FUNCTION_BLOCK FB_DriveInverter EXTENDS FB_DriveReverse IMPLEMENTS I_DriveInverter;
VAR
	_stInverter : ST_Inverter;
			
END_VAR

VAR_STAT
	_nInstances		: INT;		// Counter of created Instances
END_VAR

PROPERTY DeviceData : ST_Inverter
GET
// Dane pobierane i ustawiane podczas obsługi Invertera przez ModbusRtu
DeviceData := _stInverter;
END_GET
END_PROPERTY

METHOD FB_init : BOOL
VAR_INPUT
	bInitRetains : BOOL; // if TRUE, the retain variables are initialized (warm start / cold start)
	bInCopyCode : BOOL;  // if TRUE, the instance afterwards gets moved into the copy code (online change)
	bDeviceId		 : BYTE;	
END_VAR
THIS^._stInverter.bDeviceID := bDeviceID;

//count of FB Instances and setting int Array of Interface variables. Assign an object to an interface variable
// The array of interface variable must be global
_nInstances := _nInstances + 1;
Itf.aItfDriveInverter[_nInstances] := THIS^;
END_METHOD

PROPERTY InstanceCounter : INT
GET
InstanceCounter := _nInstances;
END_GET
END_PROPERTY

METHOD Reset : BOOL
VAR_INPUT
END_VAR


// Set reset Command
THIS^._stInverter.eControl := eReset;
END_METHOD

METHOD SetSpeed : BOOL
VAR_INPUT
	_speed	: REAL;
END_VAR
//Conversion speed to Inverter register Word 
THIS^._stInverter.rSpeed := REAL_TO_WORD(_speed * 10);
END_METHOD

METHOD StatusState : STRING
VAR_INPUT
END_VAR
//Override
END_METHOD

METHOD SwitchOff : BOOL
VAR_INPUT
END_VAR
//Override  send "stop" command to modbus block

THIS^._stInverter.eControl := eReady; (*Set Ready Command (its mean stop inverter)*)
END_METHOD

METHOD SwitchOn : BOOL
VAR_INPUT
END_VAR
//Override  send "start" command to Modbus block


THIS^._stInverter.eControl := eStart; (*Set Ready Command (its mean stop inverter)*)
END_METHOD

METHOD SwitchReverseOff : BOOL
//Override  send "reverse" stop command to Modbus block


THIS^._stInverter.eControl := eReady; (*Set Ready Command (its mean stop inverter)*)
END_METHOD

METHOD SwitchReverseOn : BOOL
//Override  send "reverse" start command to Modbus block



THIS^._stInverter.eControl := eRevers; (*Set Ready Command (its mean stop inverter)*)
END_METHOD

END_FUNCTION_BLOCK

(* stored: Version 1.1.0.1, ProductVersion 3.1.4024.12
   POU FB_DriveInverter: Id {3b50846e-6152-4329-9a31-34ca455c4ec3}, SpecialFunc None
   Property DeviceData: Id {3e807e5e-639e-4fa9-8d07-f9104c80c7b0}
   Get Get: Id {af55e23d-2c03-48d1-be07-ab42e8eb159a}
   Method FB_init: Id {6d280acc-97e0-46f6-b62b-83d083551f4d}
   Property InstanceCounter: Id {f4d36832-326f-4423-aa7e-3d50b61c3b37}
   Get Get: Id {2101744b-ceb3-42e7-aebf-174bb4d76333}
   Method Reset: Id {64b64920-6b0e-4b95-82d2-e242fdbecf20}
   Method SetSpeed: Id {ffbd82cf-721f-4d5f-82e9-2001d00f4e60}
   Method StatusState: Id {b2fd76c3-f710-4a43-a23d-38a510ede9d2}
   Method SwitchOff: Id {2f65f00a-f656-42e9-8005-44be524860e7}
   Method SwitchOn: Id {76402309-67ef-4b97-8c86-4d742fe7270a}
   Method SwitchReverseOff: Id {e2abbc87-bf0f-449b-b617-af2f148cc1f4}
   Method SwitchReverseOn: Id {fa8df555-f63f-4670-adb2-e7de773a03c4} *)
